FUNCTION_BLOCK AddMover_TestSuite
VAR
	ThisTestSuite : TestSuite<TestSuiteParameter.MaxTestCount>('C:\ProgramData\Beckhoff\TwinCAT\3.1\Boot\AddMover_Tests.xml') := (TestSuiteName := 'AddMOver Test Suite');
END_VAR

TaskAcceptsMover_Test();
TaskAcceptsValidCAGroup();
TaskRejectsCyclewithNoCAGroup_Test();
TaskRejectsInvalidMover_Test();
TaskRejectsDuplicateCommand_Test();
TaskRejectsInvalidCAGroup();

METHOD TaskAcceptsMover_Test
VAR
	stubCAGroup : CollisionGroup;
	stubAxis : XtsMover;
	stubAxis1 : XtsMover;
	testMoverToGrp : AddMoverToGroupTask:= (MyCollisionGroup := stubCAGroup);
	Expected : BOOL := TRUE;
	Actual	 : BOOL;
END_VAR
IF ThisTestSuite.Test(__POUNAME()).ExecuteTest() THEN
	Actual := SUCCEEDED(testMoverToGrp.AddMover(stubAxis));
	ThisTestSuite.Test(__POUNAME()).AssertEqual(Expected, Actual);
END_IF
END_METHOD

METHOD TaskAcceptsValidCAGroup
VAR
	stubCAGroup : CollisionGroup;
	istuibCAGroup : I_CollisionGroup := stubCAGroup;
	testMoverToGrp : AddMoverToGroupTask;
	Expected : BOOL := TRUE;
	Actual	 : BOOL;
END_VAR
IF ThisTestSuite.Test(__POUNAME()).ExecuteTest() THEN
	testMoverToGrp.MyCollisionGroup := stubCAGroup;
	Actual := testMoverToGrp.MyCollisionGroup = istuibCAGroup;
	ThisTestSuite.Test(__POUNAME()).AssertEqual(Expected, Actual);
END_IF
END_METHOD

METHOD TaskRejectsCyclewithNoCAGroup_Test
VAR
	stubCAGroup : CollisionGroup;
	stubAxis : XtsMover;
	stubAxis1 : XtsMover;
	testMoverToGrp : AddMoverToGroupTask:= (MyCollisionGroup := stubCAGroup);
	Expected : BOOL := TRUE;
	Actual	 : BOOL;
END_VAR
IF ThisTestSuite.Test(__POUNAME()).ExecuteTest() THEN
	Actual := FAILED(testMoverToGrp.Cycle());
	ThisTestSuite.Test(__POUNAME()).AssertEqual(Expected, Actual);
END_IF
END_METHOD

METHOD TaskRejectsDuplicateCommand_Test
VAR
	stubCAGroup : CollisionGroup;
	stubAxis : XtsMover;
	stubAxis1 : XtsMover;
	testMoverToGrp : AddMoverToGroupTask:= (MyCollisionGroup := stubCAGroup);
	Expected : BOOL := TRUE;
	Actual	 : BOOL;
END_VAR
IF ThisTestSuite.Test(__POUNAME()).ExecuteTest() THEN
	testMoverToGrp.AddMover(stubAxis);
	Actual := FAILED(testMoverToGrp.AddMover(stubAxis1));
	ThisTestSuite.Test(__POUNAME()).AssertEqual(Expected, Actual);
END_IF
END_METHOD

METHOD TaskRejectsInvalidCAGroup
VAR
	stubCAGroup : CollisionGroup;
	iStubCAGroup : I_CollisionGroup := stubCAGroup;
	testMoverToGrp : AddMoverToGroupTask:= (MyCollisionGroup := stubCAGroup);
	Expected : BOOL := TRUE;
	Actual	 : BOOL;
END_VAR
IF ThisTestSuite.Test(__POUNAME()).ExecuteTest() THEN
	testMoverToGrp.MyCollisionGroup := 16#0;
	Actual := testMoverToGrp.MyCollisionGroup = iStubCAGroup;
	ThisTestSuite.Test(__POUNAME()).AssertEqual(Expected, Actual);
END_IF
END_METHOD

METHOD TaskRejectsInvalidMover_Test
VAR
	stubCAGroup : CollisionGroup;
	stubAxis : XtsMover;
	stubAxis1 : XtsMover;
	testMoverToGrp : AddMoverToGroupTask:= (MyCollisionGroup := stubCAGroup);
	Expected : BOOL := TRUE;
	Actual	 : BOOL;
END_VAR
IF ThisTestSuite.Test(__POUNAME()).ExecuteTest() THEN
	Actual := FAILED(testMoverToGrp.AddMover(16#0));
	ThisTestSuite.Test(__POUNAME()).AssertEqual(Expected, Actual);
END_IF
END_METHOD

END_FUNCTION_BLOCK

(* stored: Version 1.1.0.1
   POU AddMover_TestSuite: Id {e6d2eae2-d6b8-40f3-b93b-ee6358707c5b}, SpecialFunc None
   Method TaskAcceptsMover_Test: Id {76d622a8-3592-402c-963b-8fe6effd36e5}
   Method TaskAcceptsValidCAGroup: Id {3c10fd1e-0467-4752-98d7-57c24a691c09}
   Method TaskRejectsCyclewithNoCAGroup_Test: Id {67079034-a882-4395-b22e-5f8c5fbf43fc}
   Method TaskRejectsDuplicateCommand_Test: Id {caf75f25-819a-48cc-a5c7-cd789f30bab6}
   Method TaskRejectsInvalidCAGroup: Id {416b9f46-b726-406d-ae68-ebe97a7a40e7}
   Method TaskRejectsInvalidMover_Test: Id {e3b9e3da-2293-4563-b5f0-6f0df1b14381} *)
